// TIA Portal project "debugger" (V16)

(* hardware
DEVICE "PC station"  SIMATIC PC station
   slot 0: "PC station"  Rail  SIMATIC PC-Station  V1.0
      slot 125: "Stationmanager"  Station_Manager  V6.0.4
   slot 1: "IE general_1"  IE General  IE_CP  V8.2.0
   slot 3: "HMI_RT_1"  WinCC Unified Scada RT  6AV2 155-xxxxx-xxxx  16.0.0.0
*)

(* ===== HMI "HMI_RT_1" =====

HMI tags "Default tag table"
   "gaugeTag" : Int, internal

text list "SystemTextList_ConfigErrorAlarmTextLibrary_1": 1 'NameService configuration error: Implicit deletion - Subelement instance @6%s@ must be deleted explicitly'; 2 'NameService configuration error: Implicit deletion - Alias/Format/Unit instance @6%s@ must be deleted explicitly'

text list "SystemTextList_ConfigErrorAlarmTextLibrary_2": 1 'EvDpManager::cleanupDeletedDatapoint - alert handler config is deleted implicitly for deleted datapoint, @3%s@'; 2 'EvDpManager::cleanupDeletedDatapoint - alert handler config is deleted implicitly but still has overrides, @3%s@'; 3 'EvDpManager::cleanupDeletedDatapoint - default value config is deleted implicitly for deleted datapoint, @3%s@'; 4 'EvDpManager::cleanupDeletedDatapoint - default value config is deleted implicitly but still has overrides, @3%s@'; 5 'EvDpManager::cleanupDeletedDatapoint - initial value config is deleted implicitly for deleted datapoint, @3%s@'; 6 'EvDpManager::cleanupDeletedDatapoint - initial value config is deleted implicitly but still has overrides, @3%s@'; 7 'EvDpManager::cleanupDeletedDatapoint - distribution config is deleted implicitly for deleted datapoint, @3%s@'; 8 'EvDpManager::cleanupDeletedDatapoint - distribution config is deleted implicitly but still has overrides, @3%s@'; 9 'EvDpManager::cleanupDeletedDatapoint - rangeCheck config is deleted implicitly for deleted datapoint, @3%s@'; 10 'EvDpManager::cleanupDeletedDatapoint - rangeCheck config is deleted implicitly but still has overrides, @3%s@'

text list "SystemTextList_ConfigErrorAlarmTextLibrary_3": 1 'DpType has been deleted but there is still a type config defined for the type node, @3%s@'; 2 'DpTypeNode has been deleted in DpType but there is still a type config defined for the element, @3%s@'

text list "SystemTextList_ConfigErrorAlarmTextLibrary_4": 2 'HmiCycle - @6%s@ does not exist'; 3 'HmiAlarm - @6%s@ already exists'; 4 'HmiTag - Address @6%s@ was rejected'; 1 'HmiConnection - @6%s@ does not exist'; 5 'HmiTag - Acquisition mode @6%s@ is not supported by CHROM'; 6 'HmiCycle - @6%s@ deleted, but associated HmiTags exist'; 7 'HmiConnection - @6%s@ deleted, but associated HmiTags exist'; 8 'HmiTag - SelectorTag @6%s@ was rejected'; 9 'HmiTag - SelectorTag @6%s@ has an invalid value'; 0 'Connection could not be established - @6%s@'; 65638 'Connection could not be established - @6%s@'; 65639 'Connection lost - @6%s@'; 65640 'Connection lost on HMI side - @6%s@'; 65641 'Connection lost on PLC side - @6%s@'; 65541 'Connection could not be established - Open timed out - @6%s@'; 65542 'Connection Disturbed - @6%s@'; 65543 'Connection closed on HMI side - HmiConnection @5%s@ is changed'; 65544 'Connection closed on HMI side - Driver attribute is changed - Connection @5%s@'

text list "SystemTextList_ConfigErrorAlarmTextLibrary_5": 1 'HmiConnection - HeartbeatCycle must be lower than HeartbeatResponse'; 2 'HmiConnection - Cyclic Services are configured, but not supported on the target device'; 3 'HmiConnection - Change Driven Read is configured, but not supported on the target device'; 4 'HmiTag - The address @6%s@ does not exist in the PLC'; 5 'HmiTag - The default transformation type for address @6%s@ could not be determined'; 6 'HmiTag - Illegal transformation type.'; 7 'HmiCycle - Cannot be used, transformation is unsupported on HmiCycle'; 4096 'HmiConnection - Address version @6%s@ is not supported yet'; 4097 'HmiConnection - Profibus Addresses are not supported yet'; 4098 'HmiConnection - Softbus Addresses are not supported yet'; 4099 'HmiConnection - Address Type @6%s@ is not supported'; 4100 'HmiConnection - Invalid named connection @6%s@. AccessPoint is ignored'; 4101 'HmiConnection - Routed addresses are not supported. RouteHop @6%s@ won't be used.'; 4102 'HmiConnection - Routed addresses are not supported. RouteNet @6%s@ won't be used.'; 4103 'HmiConnection - Invalid IP address @6%s@'; 4104 'HmiConnection - Invalid named connection @6%s@. Format is supposed to be >VMD</>Connection<'; 4105 'HmiConnection - Invalid named connection @6%s@. VMD too long. At most 24 characters are allowed.'; 4106 'HmiConnection - Invalid named connection @6%s@. Connection too long. At most 32 characters are allowed.'; 4107 'HmiConnection - Rack number @6%s@ is out of range (0..7)'; 4108 'HmiConnection - Invalid named connection @6%s@. Rack is ignored'; 4109 'HmiConnection - Slot number @6%s@ is out of range (1..32)'; 4110 'HmiConnection - Invalid named connection @6%s@. Slot is ignored'; 4111 'Connection could not be established - Maximum number of possible connections (@6%s@) reached'; 4112 'Connection broken - No life sign received in last @6%s@ ms.'; 4113 'Connection could not be established - @5%s@'; 4114 'Connection could not be established - The provided address @6%s@ cannot be used'; 4115 'Connection could not be established - Invalid address @6%s@'; 4116 'Connection could not be established - @5%s@'

text list "SystemTextList_ConfigErrorAlarmTextLibrary_6": 1 'Connection not established - Application instance certificate not configured'; 2 'Connection not established - Server rejected client certificate - OPC UA status code @5%s@'; 3 'Connection not established - Internal certificate store problem - OPC UA status code @5%s@'; 4 'Connection not established - Loading application instance certificate failed - OPC UA status code @5%s@'; 5 'Connection not established - Server has not provided certificate. @5%s@'; 6 'Connection not established - Server certificate validation failed - OPC UA status code @5%s@'; 7 'Connection was closed - Alarm synchronization failed - OPC UA status code @5%s@'; 8 'Connection was closed - Alarm/Event subscription failed due to server operation count limit exceeded'; 9 'Connection was closed - Alarm/Event subscription failed due to server subscription count limit exceeded'; 10 'Connection not established - Server reported license problem - OPC UA status code @5%s@'; 11 'Connection not established - Maximum Number of Server Sessions reached'; 12 'Connection not established - Inconsistent security configuration - @5%s@'; 13 'Connection not established - The provided address @5%s@ cannot be used'; 14 'Connection not established - OPC UA status code @5%s@'; 15 'The connection was lost - OPC UA server was shut down'; 16 'The connection was lost - No life sign received in last @5%s@ milliseconds'; 17 'Connection was closed - OPC UA Server in maintenance'; 18 'Connection not established - Invalid authentication configuration with Authentication Mode - @5%s@'; 19 'Connection not established - User could not be authenticated - OPC UA status code @5%s@'; 20 'Connection not established - Anonymous connection not allowed by server - OPC UA status code @5%s@'; 21 'Connection not established - Certificate problem. Failed to write security relevant file to directory @5%s@'; 22 'Connection not established - Certificate problem. Unexpected file in certificate directory @5%s@ cannot be removed'; 23 'Connection not established - User could not be authenticated - empty userID and password configured'; 24 'Connection not established - Length of configured server certificate exceeded limit. @5%s@'; 25 'Connection not established - Configured @5%s@ has zero length'; 26 'Connection not established - Configured @5%s@ has unexpected format'; 27 'Connection not established - Cannot read endpoints from server. OPC UA status code @5%s@'; 28 'Connection not established - No endpoints found for server. @5%s@'; 29 'Connection not established - Application instance certificate not found.'; 30 'Connection not established - Unexpected format of certificate @5%s@'; 31 'Connection not established - Unexpected format of revocation list @5%s@'; 101 'HmiTag - Provided address @6%s@ does not exist in the server'; 103 'HmiTag - Provided address @6%s@ is not accessible'; 104 'HmiTag - Acquisition Mode not supported for provided address @6%s@'; 201 'HmiAlarm - Provided address @6%s@ does not exist in the server'; 202 'HmiAlarm - Provided address @6%s@ cannot be used because the area filter provided is not an OPC UA event notifier'; 203 'HmiAlarm - Provided address @6%s@ cannot be used because the area filter provided does not exist in the server'; 204 'HmiAlarm - Provided address @6%s@ cannot be used because it is not an OPC UA event type'; 205 'HmiAlarm - Provided address @6%s@ cannot be used because the OPC UA condition type is not supported'; 206 'HmiAlarm - Provided address @6%s@ cannot be used because the event type provided does not exist in the server'; 207 'HmiAlarm - Acquisition Mode value not supported for provided address @6%s@'; 301 'Provided address @6%s@ cannot be used because it is missing version'; 302 'Provided address @6%s@ cannot be used because it contains invalid version'; 303 'Provided address @6%s@ cannot be used because it has invalid count of separators '$''; 304 'Provided address @6%s@ cannot be used because the address kind is invalid'; 305 'Unsupported version @6%s@ of Address'; 401 'Unexpected OPC UA Server response: @6%s@'

text list "SystemTextList_ConfigErrorAlarmTextLibrary_7": 1 'AlarmAnnunciator - Invalid condition string for annunciator @6%s@'; 2 'AlarmAnnunciator - Invalid state tag and bit for annunciator @6%s@'; 3 'AlarmAnnunciator - Invalid silence control tag and bit for annunciator @6%s@'

text list "SystemTextList_ConfigErrorAlarmTextLibrary_8": 1 'TagLogging configuration error: implicit deletion - LoggingTag instance @6%s@ should be deleted but has overrides'

text list "SystemTextList_ConfigErrorAlarmTextLibrary_9": 1 ''; 2 'Restart of the runtime is required!'; 3 'Eject and insert of correct media is required!'

text list "SystemTextList_S7PlusAlarmTextListCollection_1": 4096 'Connection lost on PLC side - @5%s@'; 4097 'Connection lost on HMI side - @5%s@'; 4098 'Maximum number of connections exceeded - @5%s@'; 4099 'Out of resources on PLC - @5%s@'; 4100 'Legitimation failed, invalid or missing password - @5%s@'; 4101 'Open request failed - @5%s@'; 4102 'Cannot connect to PLC - @5%s@'; 4103 'Open request could not be sent'
*)